{attribute 'qualified_only'}
{attribute 'strict'}
TYPE CmdRobot :
(
	noCmd                :=0,
	Cmd_GoHome           :=1,//1=回原点 
	Cmd_GoAutoProcesses  :=2//到取料位
)INT;
END_TYPE

(* stored: Version 1.1.0.1, ProductVersion 3.1.4024.9
   DUT CmdRobot: Id {6912cb9a-b56c-431f-854a-86a6871ed767} *)
